Universal Robots PolyScope program: firsttask.urp

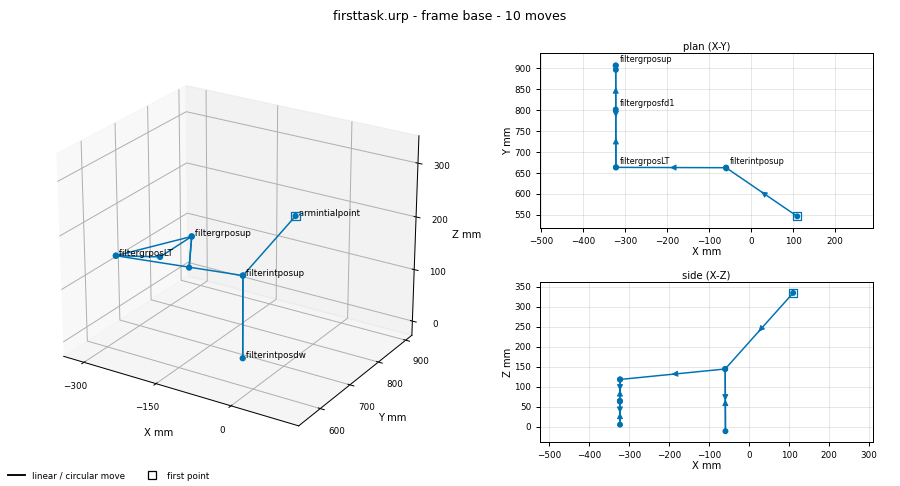
[picture p0: tool path of firsttask.urp in frame base, 10 of 10 moves have a stored position in this frame; points joined in program order, loops and branches not executed]
Program firsttask (installation=default directory=/programs/usbdisk createdIn=5.14.6 lastSavedIn=5.14.6 robotSerialNumber=20195002010)
Calibrated DH parameters: a=[0.000102, -0.601263, -0.549927, 0.000052, -0.000116, 0]; d=[0.180865, -56.180042, 109.263409, -52.909159, 0.11991, 0.115616]; alpha=[1.571117, -0.002043, -0.002909, 1.571266, -1.570859, 0]; deltaTheta=[0, 0.188632, 5.82082, 0.273737, -0.000003, 0]
InitVariablesNode
Robot Program (runOnlyOnce=true)
  MoveL speed 100 mm/s, acceleration 1200 mm/s^2 (useActiveTCP=true) feature=Base
    URCap RG Grip (OnRobot, OnRobot A/S) dataModel(rg-target-force=40.0, rg-target-width=0.032)
    Waypoint armintialpoint: motionParameters(nextMotionTime=2); TCP in base x=110.226 y=546.613 z=333.908 mm, rx=-2.1393 ry=2.205 rz=0.0002 rad; joints [97.614, -82.829, -130.419, -54.375, -273.281, 99.291] deg; TCP offset x=0 y=0 z=30.6 mm, rx=0 ry=0 rz=0 rad
    Waypoint filterintposup: TCP in base x=-59.556 y=662.633 z=143.857 mm, rx=2.0912 ry=-2.332 rz=-0.123 rad; joints [109.138, -92.637, -121.266, -52.097, -268.007, 115.453] deg; TCP offset x=0 y=0 z=223.4 mm, rx=0 ry=0 rz=0 rad
    Waypoint filterintposdw: TCP in base x=-58.916 y=661.024 z=-11.625 mm, rx=2.091 ry=-2.3321 rz=-0.123 rad; joints [109.141, -104.704, -128.109, -33.188, -267.982, 115.435] deg; TCP offset x=0 y=0 z=223.1 mm, rx=0 ry=0 rz=0 rad
    URCap RG Grip (OnRobot, OnRobot A/S) dataModel(rg-target-force=40.0, Variable(key=on_return, variable(name=on_return)))
    Waypoint filterintposup: TCP in base x=-59.556 y=662.633 z=143.857 mm, rx=2.0912 ry=-2.332 rz=-0.123 rad; joints [109.138, -92.637, -121.266, -52.097, -268.007, 115.453] deg; TCP offset x=0 y=0 z=223.4 mm, rx=0 ry=0 rz=0 rad
    MoveL speed 250 mm/s, acceleration 1200 mm/s^2 (useActiveTCP=true) feature=Base
      Waypoint filtergrposLT: TCP in base x=-322.234 y=663.457 z=117.687 mm, rx=2.0911 ry=-2.3321 rz=-0.1228 rad; joints [129.209, -100.129, -115.573, -49.826, -269.515, 135.473] deg; TCP offset x=0 y=0 z=226.9 mm, rx=0 ry=0 rz=0 rad
      Waypoint filtergrposfd1: TCP in base x=-322.729 y=801.549 z=62.5 mm, rx=2.0892 ry=-2.3302 rz=-0.1006 rad; joints [123.028, -114.089, -102.745, -49.614, -268.992, 129.307] deg
      Waypoint filtergrposup: TCP in base x=-322.776 y=906.365 z=63.902 mm, rx=2.0891 ry=-2.3302 rz=-0.1006 rad; joints [119.471, -121.813, -90.12, -54.596, -268.797, 125.76] deg
      Waypoint filtergrposdw: TCP in base x=-322.454 y=896.177 z=4.705 mm, rx=2.089 ry=-2.3302 rz=-0.1005 rad; joints [119.767, -124.212, -93.247, -49.067, -268.806, 126.048] deg
      URCap RG Grip (OnRobot, OnRobot A/S) dataModel(rg-target-force=40.0, rg-target-width=0.03)
      Waypoint filtergrposup: TCP in base x=-322.776 y=906.365 z=63.902 mm, rx=2.0891 ry=-2.3302 rz=-0.1006 rad; joints [119.471, -121.813, -90.12, -54.596, -268.797, 125.76] deg
      Waypoint filtergrposLT: TCP in base x=-322.234 y=663.457 z=117.687 mm, rx=2.0911 ry=-2.3321 rz=-0.1228 rad; joints [129.209, -100.129, -115.573, -49.826, -269.515, 135.473] deg
